{attribute 'linkalways'} 
{attribute 'no_explicit_call' := 'This FB is a CLASS and must be accessed using methods or properties'}
{attribute 'enable_dynamic_creation'}
FUNCTION_BLOCK Node_F_VN_MatchTemplateWalshExp EXTENDS VisionNode
VAR
    ipSrcImage : _ITcVnImage;
    ipTemplateImage : _ITcVnImage;
	nProjections : _UDINT(10);
	eOptions : _ETcVnMatchTemplateWalshOptions(ETcVnMatchTemplateWalshOptions.TCVN_MTWO_NONE);
	nRotations : _UDINT(1);
    ipResultImage : _ITcVnImage;
    hrPrev : _HRESULT(S_OK);
	hresult : _HRESULT(S_OK);
END_VAR

METHOD PUBLIC  Clone : I_Node
VAR
	pNode : POINTER TO Node_F_VN_MatchTemplateWalshExp;
END_VAR
pNode := __NEW(Node_F_VN_MatchTemplateWalshExp);
Clone := pNode^;
END_METHOD

METHOD FB_init : BOOL
VAR_INPUT
	bInitRetains : BOOL; // if TRUE, the retain variables are initialized (warm start / cold start)
	bInCopyCode : BOOL;  // if TRUE, the instance afterwards gets moved into the copy code (online change)
END_VAR
AddInput('ipSrcImage', ipSrcImage);
AddInput('ipTemplateImage', ipTemplateImage);
AddInput('nProjections', nProjections);
AddInput('eOptions', eOptions);
AddInput('nRotations', nRotations);
AddInput('hrPrev', hrPrev);
AddOutput('ipResultImage', ipResultImage);
AddOutput('hresult',hresult);
END_METHOD

METHOD PROTECTED OnExecute
hresult.Value := F_VN_MatchTemplateWalshExp(
    ipSrcImage := ipSrcImage.Value,
    ipTemplateImage := ipTemplateImage.Value,
	ipResultImage := ipResultImage.Value,
	nProjections := nProjections.Value,
	eOptions := eOptions.Value,
	nRotations := nRotations.Value,	
	hrPrev:= hrPrev.Value);
END_METHOD

METHOD PUBLIC PreExecutionCheck
VAR_INPUT
	Check : I_PreExecutionChecks;
END_VAR
Check.IsTrue(ipSrcImage.IsValid, 'ipSrcImage must contain an image');
Check.IsTrue(ipSrcImage.IsPixelDepth(8), 'ipSrcImage must be 8 or 32 bit pixel depth');
Check.IsTrue((ipSrcImage.HasChannelCount(1) OR ipSrcImage.HasChannelCount(3)), 'ipSrcImage must contain 1 or 3 channels');

Check.IsTrue((nRotations.Value = 1 OR nRotations.Value = 2 OR nRotations.Value = 4), 'nRotations must be 1, 2 or 4');

Check.IsTrue(ipTemplateImage.IsValid, 'ipTemplateImage must contain an image');
Check.IsTrue(ImagesHaveMatchingPixelFormats(ipSrcImage.Value, ipTemplateImage.Value), 'ipTemplateImage must have same pixel depth as ipSrcImage');
Check.IsTrue(ImagesHaveMatchingChannels(ipSrcImage.Value, ipTemplateImage.Value), 'ipTemplateImage must have same amount of channels as ipSrcImage');
Check.IsTrue(IsTemplateImageSmallerThanSourceImage(ipSrcImage.Value, ipTemplateImage.Value), 'ipTemplateImage must be smaller than ipSrcImage');
END_METHOD

END_FUNCTION_BLOCK

(* stored: Version 1.1.0.1, ProductVersion 3.1.4026.13
   POU Node_F_VN_MatchTemplateWalshExp: Id {6b62dd46-89cc-03da-2c0c-98c2fbf3b3ec}, SpecialFunc None
   Folder Constructor: Id {3c15799c-26fb-013c-0cf0-fbfa5e1db58f}
   Method Clone: Id {d00f8e9d-6e85-0b3e-20fd-6e8756844721}
   Method FB_init: Id {971a4b85-51b2-0f81-3877-101d2df5dfff}
   Method OnExecute: Id {00babf95-0810-0ea4-2080-493d04983d19}
   Method PreExecutionCheck: Id {f2148062-8431-0634-0d21-cc907bc74f8b} *)
